{attribute 'qualified_only'}
{attribute 'strict'}
TYPE E_SDSFaceState :
(
    UNKNOWN := 0,
    FACE_TRANSFER_ARM := 1,
    FACE_SIDE_PORT := 2
) UINT;
END_TYPE

(* stored: Version 1.1.0.1
   DUT E_SDSFaceState: Id {6d8a622b-81c8-4cf8-adfa-d15a25824ce2} *)
